// Mitsubishi GX Works2 project: 0129 deco기초   PLC: Q03UDV

PROGRAM MAIN
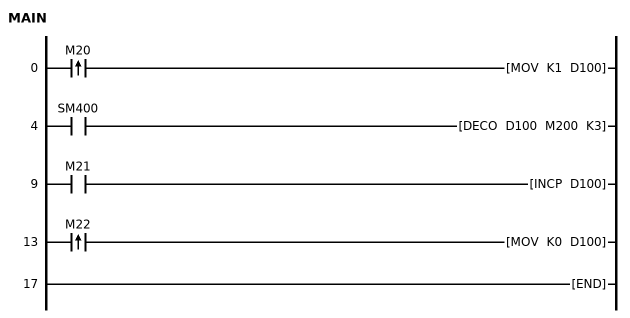
0     LDP     M20
      MOV     K1 D100
4     LD      SM400
      DECO    D100 M200 K3
9     LD      M21
      INCP    D100
13    LDP     M22
      MOV     K0 D100
17    END
END_PROGRAM
